FUNCTION_BLOCK TIMER_SIMULATION
  {SET_ATTRIBUTE(OpcUa, SERVICE)}
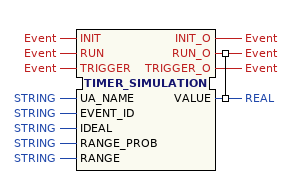
  EVENT_INPUT
    INIT;
    RUN;
    TRIGGER;
  END_EVENT
  EVENT_OUTPUT
    INIT_O;
    RUN_O WITH VALUE;
    TRIGGER_O;
  END_EVENT
  VAR_INPUT
    UA_NAME : STRING; {SET_ATTRIBUTE(OpcUa, Constant)}
    EVENT_ID : STRING; {SET_ATTRIBUTE(OpcUa, Constant)}
    IDEAL : STRING; {SET_ATTRIBUTE(OpcUa, Constant)}
    RANGE_PROB : STRING; {SET_ATTRIBUTE(OpcUa, Constant)}
    RANGE : STRING; {SET_ATTRIBUTE(OpcUa, Constant)}
  END_VAR
  VAR_OUTPUT
    VALUE : REAL; {SET_ATTRIBUTE(OpcUa, Variable)}
  END_VAR
END_FUNCTION_BLOCK
